// TIA Portal V17 export
// export: Created 2022-10-14T12:26:29.0320906Z, ExportSetting WithDefaults, DisplayName Totally Integrated Automation Portal, DisplayVersion V17 Update 4, DisplayName TIA Portal Openness, DisplayVersion V17 Update 4, DisplayName TIA Portal Version Control Interface, DisplayVersion V17, DisplayName SINAMICS Startdrive Advanced, DisplayVersion V17 Update2, DisplayName SINAMICS Startdrive G130, G150, S120, S150, SINAMICS MV, S210, DisplayVersion V17 Update2, DisplayName SINAMICS Startdrive G110M, G120, G120C, G120D, G120P, G115D, DisplayVersion V17 Update2, DisplayName STEP 7 Professional, DisplayVersion V17 Update 4, DisplayName STEP 7 Safety, DisplayVersion V17, DisplayName WinCC Advanced / Unified PC, DisplayVersion V17 Update 4
FUNCTION_BLOCK "Speed_KreisBahn"   // FB2, FBD
{ S7_Optimized_Access := 'TRUE' }
VERSION : 0.1
// stored: AutoNumber true, IsIECCheckEnabled false, IsRetainMemResEnabled false, MemoryReserve 100, SetENOAutomatically false, UDAEnableTagReadback false
   VAR_INPUT
      Speed : Real;
      Zeit { ExternalAccessible := 'False'; ExternalVisible := 'False'; ExternalWritable := 'False'} : Timer;
   END_VAR
   VAR_OUTPUT
      X_Pos : Int;
      Y_Pos : Int;
   END_VAR
   VAR
      Richtung : Bool;
      Time_1 : S5Time;
      HM_2 : Bool;
      i : Int;
   END_VAR
   VAR_TEMP
      H_Speed : Real;
      Norm_Real : Real;
      Scale_Int : Int;
      HInt : Int;
      HM_1 : Time;
   END_VAR
   VAR_TEMP   // added for the SCL form of the ladder/FBD networks
      _w1 : Bool;
      _s5time1 : S5Time;
   END_VAR
BEGIN

REGION Network 1
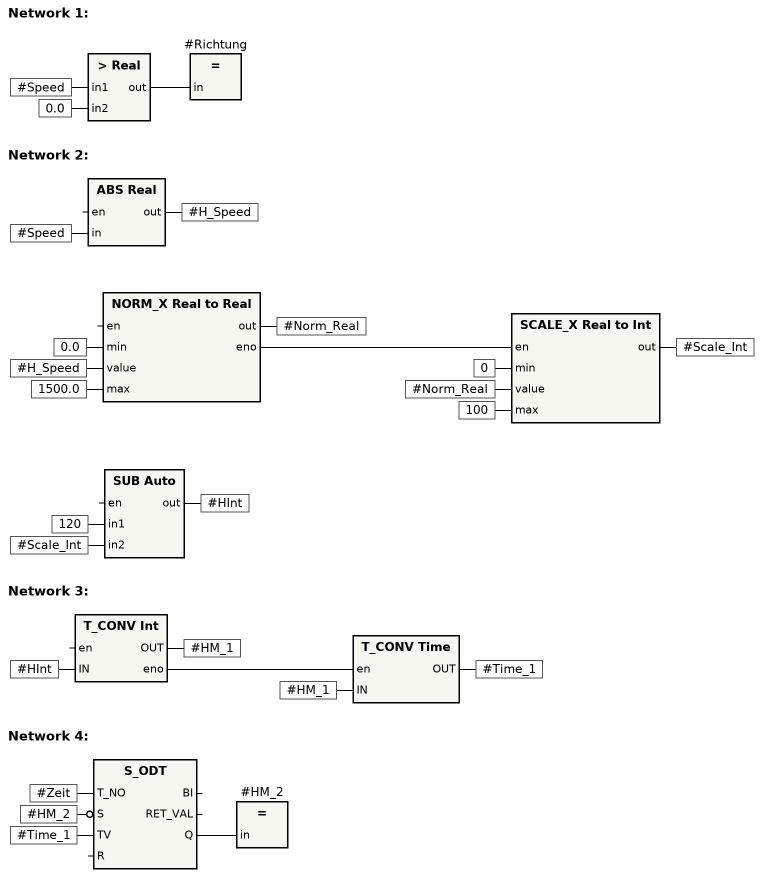
   #Richtung := #Speed > 0.0;
END_REGION

REGION Network 2
   #H_Speed := ABS(#Speed);
   #Norm_Real := NORM_X(MIN := 0.0, VALUE := #H_Speed, MAX := 1500.0);
   #Scale_Int := SCALE_X(MIN := 0, VALUE := #Norm_Real, MAX := 100);
   #HInt := 120 - #Scale_Int;
END_REGION

REGION Network 3
   T_CONV(IN := #HInt, OUT => #HM_1, ENO => #_w1);
   IF #_w1 THEN T_CONV(IN := #HM_1, OUT => #Time_1); END_IF;
END_REGION

REGION Network 4
   #_s5time1 := S_ODT(T_NO := #Zeit, S := NOT #HM_2, TV := #Time_1, Q => #_w1);
   #HM_2 := #_w1;
END_REGION

REGION Network 5
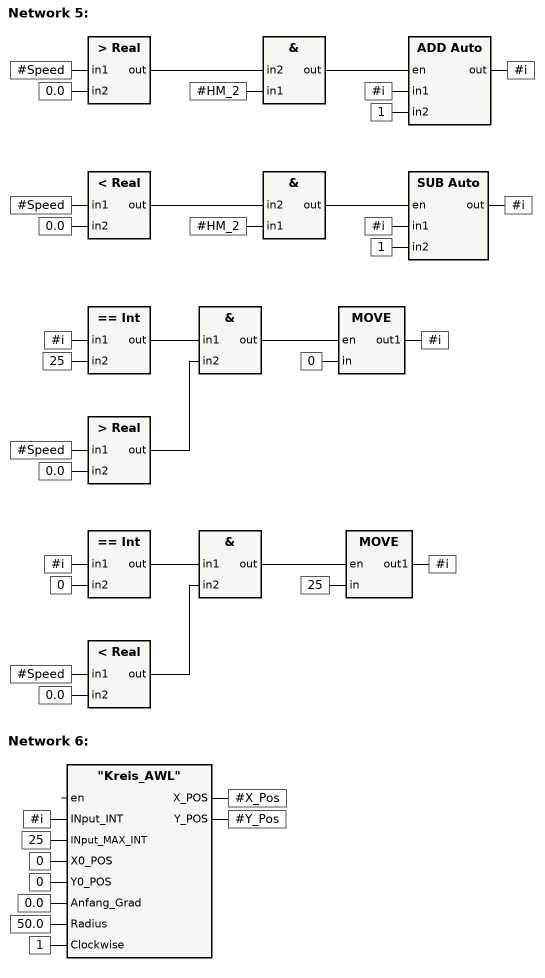
   IF (#Speed > 0.0) AND #HM_2 THEN #i := #i + 1; END_IF;
   IF (#Speed < 0.0) AND #HM_2 THEN #i := #i - 1; END_IF;
   IF (#i = 25) AND (#Speed > 0.0) THEN #i := 0; END_IF;
   IF (#i = 0) AND (#Speed < 0.0) THEN #i := 25; END_IF;
END_REGION

REGION Network 6
   "Kreis_AWL"(INput_INT := #i,
               INput_MAX_INT := 25,
               X0_POS := 0,
               Y0_POS := 0,
               Anfang_Grad := 0.0,
               Radius := 50.0,
               Clockwise := 1,
               X_POS => #X_Pos,
               Y_POS => #Y_Pos);
END_REGION
END_FUNCTION_BLOCK
